Fanuc KAREL source: kt00256.KL

-- PROVISIONAL review KL for V1013-1; original PC SHA256 e63a95573ccc2533e06031d83425aa5bbdaca8e07f125d06e088dc9bfd72c0e7
-- Incomplete behavior may be omitted. Consult companion uncertainty JSON. Do not deploy.
PROGRAM KT00256
%NOLOCKGROUP
VAR
  OUT : INTEGER
-- UNRESOLVED_DECL H1 type=002017
-- UNRESOLVED_DECL H2 type=002017
BEGIN
  -- UNRESOLVED_PC offsets 5-19; opcodes 2E,22,9D,33,B4
  -- UNRESOLVED_PC offsets 24-38; opcodes 2E,22,9D,33,B4
  -- UNRESOLVED_PC offsets 43-57; opcodes 2E,22,9D,33,B4
  -- UNRESOLVED_PC offsets 62-76; opcodes 2E,22,9D,33,B4
  -- UNRESOLVED_PC offsets 81-106; opcodes 22,9D,33,B3,22,9D,33,B3,47,23
  -- UNRESOLVED_PC offsets 111-115; opcodes 7F
END KT00256
